DATA_BLOCK "DB"
{ S7_Optimized_Access := 'true' }
    VAR
        S1_vs1: DINT;
        S2_vs2: DINT;
        S2: BOOL;
        R1_vr1: DINT;
        R2_vr2: DINT;
        R2: BOOL;
        Y1_vy1: DINT;
        Y2_vy2: DINT;
        Y2: BOOL;
        M1_vm1: DINT;
        M2_vm2: DINT;
        M2: BOOL;
        firstRun: BOOL;
    END_VAR
BEGIN
    firstRun := TRUE;
END_DATA_BLOCK
